// TIA Portal V20 export
FUNCTION_BLOCK "LER_qrHistory"   // FB195, LAD
// stored: Access Published, MemoryReserve 100, SetENOAutomatically false
   VAR_INPUT
      trigger : Bool;
      commonData : "LER_typeCommonData";
      qrData : "LER_typeQrData";
   END_VAR
   VAR_IN_OUT
      dataHistory : "LER_typeQrHistory";
   END_VAR
   VAR
      statDeleteData : "LER_typeQrHistory";
      statTrigger : Array[0..99] of Bool;
      statTonTimer { S7_SetPoint := 'True'} : Array[0..99] of TON_TIME;
      statComplete : Array[0..99] of Bool;
   END_VAR
   VAR_TEMP
      tempRetVal : Array[0..99] of Int;
   END_VAR
   VAR_TEMP   // added for the SCL form of the ladder/FBD networks
      _w1 : Bool;
   END_VAR
BEGIN

REGION Network 1
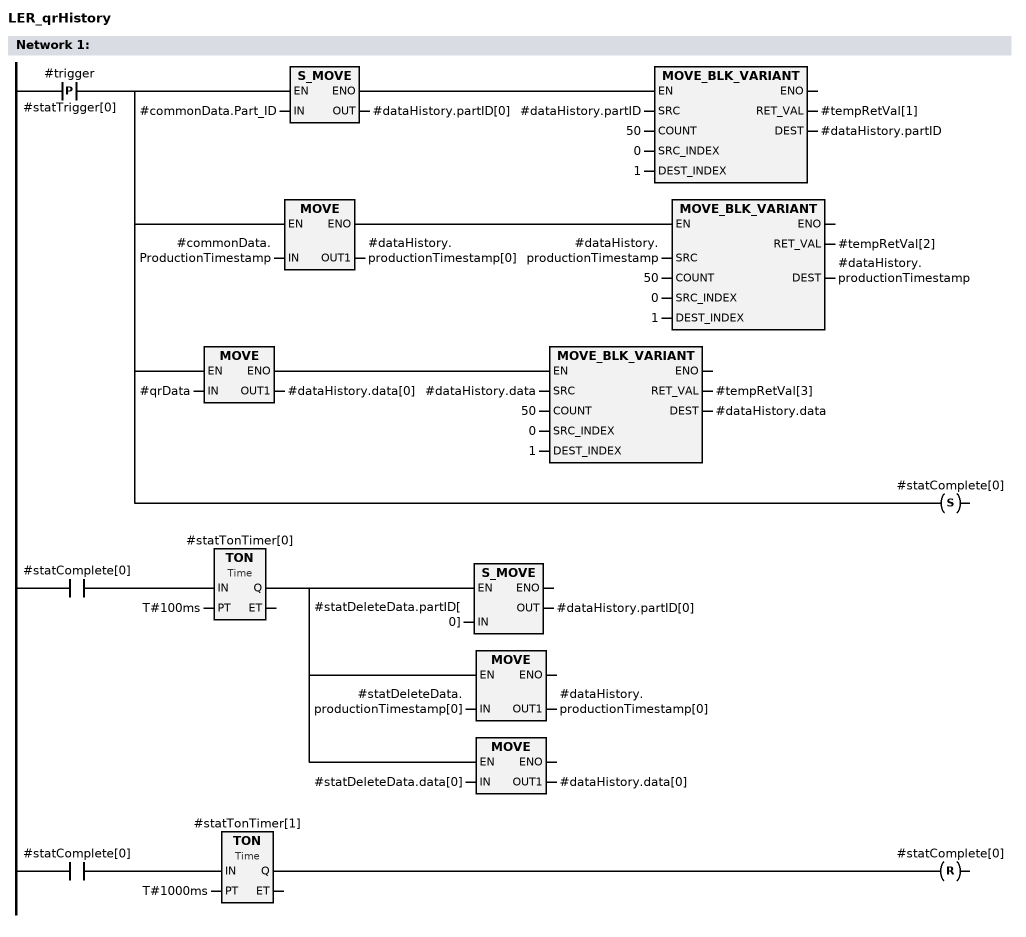
   RUNG wire#powerrail
      P_Contact(operand := #trigger, bit := #statTrigger[0])
      wire#w1
      S_Move(in := #commonData.Part_ID, out => #dataHistory.partID[0])
      MOVE_BLK_VARIANT(SRC := #dataHistory.partID, COUNT := 50, SRC_INDEX := 0, DEST_INDEX := 1, Ret_Val => #tempRetVal[1], DEST => #dataHistory.partID)
   END_RUNG
   RUNG wire#w1
      Move(in := #commonData.ProductionTimestamp, out1 => #dataHistory.productionTimestamp[0])
      MOVE_BLK_VARIANT(SRC := #dataHistory.productionTimestamp, COUNT := 50, SRC_INDEX := 0, DEST_INDEX := 1, Ret_Val => #tempRetVal[2], DEST => #dataHistory.productionTimestamp)
   END_RUNG
   RUNG wire#w1
      Move(in := #qrData, out1 => #dataHistory.data[0])
      MOVE_BLK_VARIANT(SRC := #dataHistory.data, COUNT := 50, SRC_INDEX := 0, DEST_INDEX := 1, Ret_Val => #tempRetVal[3], DEST => #dataHistory.data)
   END_RUNG
   RUNG wire#w1
      S_Coil( #statComplete[0] )
   END_RUNG
   RUNG wire#powerrail
      Contact( #statComplete[0] )
      { S7_Templates := "time_type := Time" } #statTonTimer[0].TON(pt := T#100ms, et =>)
      wire#w2
      S_Move(in := #statDeleteData.partID[0], out => #dataHistory.partID[0])
   END_RUNG
   RUNG wire#w2
      Move(in := #statDeleteData.productionTimestamp[0], out1 => #dataHistory.productionTimestamp[0])
   END_RUNG
   RUNG wire#w2
      Move(in := #statDeleteData.data[0], out1 => #dataHistory.data[0])
   END_RUNG
   RUNG wire#powerrail
      Contact( #statComplete[0] )
      { S7_Templates := "time_type := Time" } #statTonTimer[1].TON(pt := T#1000ms, et =>)
      R_Coil( #statComplete[0] )
   END_RUNG
   // the same network as SCL:
   #_w1 := #trigger AND NOT #statTrigger[0];   // rising edge of #trigger
   #statTrigger[0] := #trigger;
   IF #_w1 THEN
       #dataHistory.partID[0] := #commonData.Part_ID;
       #tempRetVal[1] := MOVE_BLK_VARIANT(SRC := #dataHistory.partID,
                               COUNT := 50,
                               SRC_INDEX := 0,
                               DEST_INDEX := 1,
                               DEST => #dataHistory.partID);
       #dataHistory.productionTimestamp[0] := #commonData.ProductionTimestamp;
       #tempRetVal[2] := MOVE_BLK_VARIANT(SRC := #dataHistory.productionTimestamp,
                               COUNT := 50,
                               SRC_INDEX := 0,
                               DEST_INDEX := 1,
                               DEST => #dataHistory.productionTimestamp);
       #dataHistory.data[0] := #qrData;
       #tempRetVal[3] := MOVE_BLK_VARIANT(SRC := #dataHistory.data,
                               COUNT := 50,
                               SRC_INDEX := 0,
                               DEST_INDEX := 1,
                               DEST => #dataHistory.data);
       #statComplete[0] := TRUE;
   END_IF;
   #statTonTimer[0].TON(IN := #statComplete[0], PT := T#100ms);
   IF #statTonTimer[0].Q THEN
       #dataHistory.partID[0] := #statDeleteData.partID[0];
       #dataHistory.productionTimestamp[0] := #statDeleteData.productionTimestamp[0];
       #dataHistory.data[0] := #statDeleteData.data[0];
   END_IF;
   #statTonTimer[1].TON(IN := #statComplete[0], PT := T#1000ms);
   IF #statTonTimer[1].Q THEN #statComplete[0] := FALSE; END_IF;
END_REGION
END_FUNCTION_BLOCK
